// TwinCAT 3 PLC project WinchCylControl
// ProgramVersion: 3.1.4023.0
// libraries:
//   Tc2_Standard, * (Beckhoff Automation GmbH)
//   Tc2_System, * (Beckhoff Automation GmbH)
//   Tc3_Module, * (Beckhoff Automation GmbH)
// project tree:
//   FunctionBlocks/ FB_Encoder.TcPOU, FB_JoystickInputScaling.TcPOU, FB_ValveOutput.TcPOU
//   Inputs/ G_InputList.TcGVL, ST_ControlBoxInputs.TcDUT, ST_CylinderInputs.TcDUT, ST_JoystickScaling.TcDUT, ST_WinchInputs.TcDUT
//   MotionControl/ Path_signal_gen.TcPOU, P_MotionxControl.TcPOU
//   MotionControl/PID-Controllers/ Closed.TcPOU, Open0.TcPOU
//   MotionControl/Structs/ ST_MotionParameters.TcDUT, ST_Params.TcDUT, ST_PathParameters.TcDUT, ST_ValveDeadBand.TcDUT
//   Outputs/ G_OutputList.TcGVL, ST_ValveOutputs.TcDUT
//   / PlcTask.TcTTO
//   POUs/ MAIN.TcPOU
//   Scaling/FBs/ FB_FlowScale.TcPOU, FB_PressureScale.TcPOU
//   Scaling/ G_ScaledIOs.TcGVL, P_Scaling.TcPOU
//   Scaling/Structs/ ST_FlowScale.TcDUT, ST_ScaledCylinderInputs.TcDUT, ST_ScaledWinchInputs.TcDUT
// real-time tasks:
//   TASK PlcTask: cycle T#10ms, priority 20, ADS port 350

CONFIGURATION WinchCylControl
    RESOURCE PLC ON TwinCAT3
        TASK PlcTask(INTERVAL := T#10ms, PRIORITY := 20);
        PROGRAM MAIN WITH PlcTask : MAIN;
    END_RESOURCE
END_CONFIGURATION

// ---- Inputs/ST_ControlBoxInputs.TcDUT
TYPE ST_ControlBoxInputs :
STRUCT
	bAutoMode AT %I* : BOOL;
	bManualMode AT %I*: BOOL;
	bStartButton AT %I*: BOOL;
	bStopButton AT %I* : BOOL; 
	bTopSwitch AT %I*: BOOL; 
	nJoyX : INT;
	nJoyY : INT; 
END_STRUCT
END_TYPE

// ---- Inputs/ST_CylinderInputs.TcDUT
TYPE ST_CylinderInputs :
STRUCT
	fPistonPressure : INT;
	fRodPressure : INT; 
	fCylinderPosition : LREAL; 
END_STRUCT
END_TYPE

// ---- Inputs/ST_JoystickScaling.TcDUT
TYPE ST_JoystickScaling :
STRUCT
	fMaxInputVal : LREAL := 20509.0;
	fMinInputVal : LREAL := 11787.0; 
	fNeutralInputVal : LREAL := 16175.0;
	fNeutralDeadBand : LREAL := 50.0; 
	fMaxOutputVal : LREAL := 1.0;
	fMinOutputVal : LREAL := -1.0;
	fNeutralOutputVal : LREAL := 0.0;
END_STRUCT
END_TYPE

// ---- Inputs/ST_WinchInputs.TcDUT
TYPE ST_WinchInputs :
STRUCT
	fWinchInletPressure : INT;
	fWinchInletPressureSensor : INT;
	fWinchOutletPressure : INT;
	fWinchOutletPressureB1 : INT;
	fWinchDrainPressure : INT; // 40 BAR
	fWinchInletFlow : INT; 
END_STRUCT
END_TYPE

// ---- MotionControl/Structs/ST_MotionParameters.TcDUT
TYPE ST_MotionParameters :
STRUCT
	bClosedLoopStart : BOOL; 
	bOpenLoopStart : BOOL; 
	bWinchEnable : BOOL;
	bCylinderEnable : BOOL; 
END_STRUCT
END_TYPE

// ---- MotionControl/Structs/ST_Params.TcDUT
TYPE ST_Params :
STRUCT
	fEncoderOffset : LREAL := 17574.8; 
	fGBtoDrumScaling : LREAL := 0.000744309; 
END_STRUCT
END_TYPE

// ---- MotionControl/Structs/ST_PathParameters.TcDUT
TYPE ST_PathParameters :
STRUCT
	x0: LREAL := 0;
	v_0: LREAL := 0;
	x_ref: LREAL := 0.3;
	v_ref: LREAL := 0.15;
	t0: LREAL := 0;
	tRamp: LREAL := 2;
	tWait: LREAL := 2;
END_STRUCT
END_TYPE

// ---- MotionControl/Structs/ST_ValveDeadBand.TcDUT
TYPE ST_ValveDeadBand :
STRUCT
	fPosMax : LREAL := 29490.0;
	fPosMin : LREAL := 20950.0;
	fNegMax : LREAL := 18250.0;
	fNegMin : LREAL := 9830.0;
END_STRUCT
END_TYPE

// ---- Outputs/ST_ValveOutputs.TcDUT
TYPE ST_ValveOutputs :
STRUCT
	bEnable AT %I* : BOOL;
	nValveOut AT %Q* : INT;
END_STRUCT
END_TYPE

// ---- Scaling/Structs/ST_FlowScale.TcDUT
TYPE ST_FlowScale :
STRUCT
	fMaxInputValue :LREAL := 32295.0;
 	fMinInputValue :LREAL := 0.0;
 	fNeutralInputValue :LREAL := 15450;
 	fNeutralDeadband :LREAL := 50.0;
	fMaxOutputValue :LREAL := 150.0; 
	fMinOutputValue :LREAL := -150.0; 
	fNeutralOutputValue :LREAL := 0.0; 
END_STRUCT
END_TYPE

// ---- Scaling/Structs/ST_ScaledCylinderInputs.TcDUT
TYPE ST_ScaledCylinderInputs :
STRUCT
	fPistonPressureS : LREAL;
	fRodPressureS : LREAL; 
	fCylinderPositionS : LREAL; 
END_STRUCT
END_TYPE

// ---- Scaling/Structs/ST_ScaledWinchInputs.TcDUT
TYPE ST_ScaledWinchInputs :
STRUCT
	fWinchInletPressureS : LREAL;
	fWinchInletPressureSensorS : LREAL;
	fWinchOutletPressureS : LREAL;
	fWinchOutletPressureB1S : LREAL;
	fWinchDrainPressureS : LREAL; // 40 BAR
	fWinchInletFlowS : LREAL; 
END_STRUCT
END_TYPE

// ---- Inputs/G_InputList.TcGVL
{attribute 'qualified_only'}
VAR_GLOBAL
	
	stModeSelect : ST_ControlBoxInputs; 
	//bManualSelect : BOOL := ST_ControlBoxInputs.bManualMode;
	//bAutoSelect : BOOL := ST_ControlBoxInputs.bAutoMode;
	//bStart : BOOL := ST_ControlBoxInputs.bStartButton;
	//bStop : BOOL := ST_ControlBoxInputs.bStopButton;
	//bTopSwitchToggle : BOOL := ST_ControlBoxInputs.bTopSwitch;

	// Joystick
	stJoystick : ST_ControlBoxInputs; 
	//nJoyXPos : INT := ST_ControlBoxInputs.nJoyX;
	//nJoyYPos : INT := ST_ControlBoxInputs.nJoyY;

	// Cylinder, Winch and pressure inputs
	fSupplyPressure AT %Q* : LREAL;
	fReturnPressure AT %Q*: LREAL;  // 40 BAR
	
	stWinchPressure : ST_WinchInputs;
	//fWinchPressureIn AT %Q* : LREAL := ST_WinchInputs.fWinchInletPressure; // A
	//fWinchPressureSensor AT %Q* : LREAL := ST_WinchInputs.fWinchInletPressureSensor; // A1
 	//fWinchPressureOut AT %Q* : LREAL := ST_WinchInputs.fWinchOutletPressure; // B
	//fWinchPressureOutB1 AT %Q* : LREAL := ST_WinchInputs.fWinchOutletPressureB1; // B1
	
	stCylinderPressures : ST_CylinderInputs;
	//fRodSidePressure AT %Q* : LREAL := ST_CylinderInputs.fRodPressure; 
	//fBoreSidePressure AT %Q* : LREAL := ST_CylinderInputs.fPistonPressure; 
	
	// Flows
	//fWinchFlow AT %Q* : LREAL := ST_WinchInputs.fWinchInletFlow;  
	
	// Får errors her
	
END_VAR

// ---- Outputs/G_OutputList.TcGVL
{attribute 'qualified_only'}
VAR_GLOBAL
	stValveOutWinch : ST_ValveOutputs;
	stValveOutCyl : ST_ValveOutputs; 
END_VAR

// ---- Scaling/G_ScaledIOs.TcGVL
{attribute 'qualified_only'}
VAR_GLOBAL
	scaledJoyX : LREAL; 
	scaledJoyY : LREAL; 
	scaledValve : LREAL; // Valve output based on joystick input [-1...1] 1 = 29490.0, -1 = 9830
	fLoadPosition : LREAL; 
	fWinchInputsScaled : ST_ScaledWinchInputs; 
	fCylinderInputsScaled : ST_ScaledCylinderInputs; 
END_VAR

// ---- POUs/MAIN.TcPOU
PROGRAM MAIN
VAR
END_VAR

END_PROGRAM

// ---- FunctionBlocks/FB_Encoder.TcPOU
FUNCTION_BLOCK FB_Encoder
VAR_INPUT
	nRawInput : UDINT;
	stParam : ST_Params; 
END_VAR
VAR_OUTPUT
	fPosition : LREAL; 
END_VAR
VAR PERSISTENT
	nRounds : DINT;
	nRawLast : DINT;
END_VAR
VAR
	nInput : DINT;
	nTempInputDiff : DINT;
	nCount : DINT;
	nMaxValue30bit : DINT := 1073741823;
	nThreshold30Bit : DINT := nMaxValue30bit/2;
	fScale16bit : LREAL := 360.0/65535.0;
	fTempPos : LREAL; 
END_VAR

nInput := UDINT_TO_DINT(nRawInput);

nTempInputDiff := nInput - nRawLast;

IF (nTempInputDiff > nThreshold30Bit) THEN
	nRounds := nRounds -1;
END_IF

IF (nTempInputDiff < nThreshold30Bit) THEN
	nRounds := nRounds + 1;
END_IF

nCount := nInput + nRounds*nMaxValue30bit;

fPosition := DINT_TO_LREAL(nCount)*fScale16bit - stParam.fEncoderOffset;

END_FUNCTION_BLOCK

// ---- FunctionBlocks/FB_JoystickInputScaling.TcPOU
FUNCTION_BLOCK FB_JoystickInputScaling
VAR_INPUT
	bEnable : BOOL; // Start Button
	bSwitch : BOOL; // TopSwitch
	nRawInput : INT;
	stJoyInputScaling : ST_JoystickScaling; 
	
END_VAR
VAR_OUTPUT
	fNormOutputC : LREAL; // Scaled cylinder output
	fNormOutputW : LREAL; // Scaled winch output
END_VAR
VAR
	fRawInput : LREAL;
	fTempInput : LREAL;
	fTempOutput : LREAL; 
END_VAR

fRawInput := INT_TO_LREAL(nRawInput);

fTempInput := fRawInput - stJoyInputScaling.fNeutralInputVal; 

IF fTempInput > stJoyInputScaling.fNeutralDeadBand THEN
	fTempOutput := fTempInput/(stJoyInputScaling.fMaxInputVal - stJoyInputScaling.fNeutralInputVal);
ELSIF fTempInput < -stJoyInputScaling.fNeutralDeadBand THEN
	fTempOutput := fTempInput/(stJoyInputScaling.fNeutralInputVal - stJoyInputScaling.fMinInputVal); 
ELSE
	fTempOutput := 0.0;
END_IF

IF NOT (bEnable) THEN
	fNormOutputC := 0; // If startbutton is not held, no joystick output
	fNormOutputW := 0.0;
ELSIF bEnable AND NOT bSwitch THEN
	fNormOutputC := LIMIT(stJoyInputScaling.fMinOutputVal, fTempOutput, stJoyInputScaling.fMaxOutputVal); 
	fNormOutputW := 0.0; // If startbutton is held but no top switch, cylinder gets output
ELSE
	fNormOutputC := 0.0; // If startbutton AND topswitch, winch gets output
	fNormOutputW := LIMIT(stJoyInputScaling.fMinOutputVal, fTempOutput, stJoyInputScaling.fMaxOutputVal); 
END_IF

END_FUNCTION_BLOCK

// ---- FunctionBlocks/FB_ValveOutput.TcPOU
FUNCTION_BLOCK FB_ValveOutput
VAR_INPUT
	bEnable : BOOL; 
	bDeadBandCompOn : BOOL;
	stValveDeadBand : ST_ValveDeadBand;
	fNormInput : LREAL; 
END_VAR
VAR_OUTPUT
	bEnableValveOutput : BOOL;
	nOutput : INT;
END_VAR
VAR
	nOffset : INT := 19660;
	nMaxValue : INT := 29490;
	nMinValue : INT := 9830;
	nTempOutput : INT; 
END_VAR

IF bDeadBandCompOn THEN
	IF fNormInput > 0.0 THEN
		nTempOutput := LREAL_TO_INT(ABS(fNormInput*(stValveDeadBand.fPosMax - stValveDeadBand.fPosMin) + stValveDeadBand.fPosMin)); 
	ELSIF fNormInput < 0.0 THEN
		nTempOutput := LREAL_TO_INT(fNormInput*(stValveDeadBand.fNegMax - stValveDeadBand.fNegMin) - stValveDeadBand.fNegMin);
	ELSE
		nTempOutput := nOffset; 
	END_IF
	
ELSE
	IF fNormInput > 0.0 THEN
		nTempOutput := LREAL_TO_INT(ABS(fNormInput*(32767.0 - 19660.0) + 19660.0));
	ELSIF fNormInput < 0.0 THEN
		nTempOutput := LREAL_TO_INT(ABS(fNormInput*(0-19660.0) - 19660.0));
	ELSE
		nTempOutput := nOffset;		
	END_IF
END_IF

IF bEnable THEN
	nOutput := LIMIT(nMinValue, nTempOutput, nMaxValue);
	bEnableValveOutput := TRUE;
ELSE
	nOutput := nOffset;
	bEnableValveOutput := FALSE; 
END_IF

END_FUNCTION_BLOCK

// ---- MotionControl/Path_signal_gen.TcPOU
FUNCTION_BLOCK Path_signal_gen
VAR_INPUT
	x0: LREAL;
	v_0: LREAL;
	x_ref: LREAL;
	v_ref: LREAL;
	t0: LREAL;
	tRamp: LREAL;
	tWait: LREAL;
	t: LREAL;
END_VAR
VAR_OUTPUT
	x: LREAL;
	v: LREAL;
	Error: LREAL;
END_VAR
VAR
	Error_0: DINT;
	tHold: LREAL;
	x1: LREAL;
	x4: LREAL;
	a_tmp: LREAL;
	a_tmp_tmp: LREAL;
	a_tmp_0: LREAL;
	a_tmp_tmp_0: LREAL;
	a_tmp_tmp_1: LREAL;
	a_tmp_tmp_2: LREAL;
	x1_tmp: LREAL;
	x4_tmp: LREAL;
END_VAR


(* MATLAB Function: '<Root>/Path_signal_gen' *)
(* MATLAB Function 'Path_signal_gen': '<S1>:1' *)
(* '<S1>:1:3' x_SetPoint = x_ref - x0; *)
(* '<S1>:1:4' vs = v_ref; *)
(* '<S1>:1:5' slopeExt = v_0-vs; *)
(* '<S1>:1:6' slopeRetr = -vs-v_0; *)
(* '<S1>:1:8' as = vs/tRamp; *)
(* Find acceleration *)
(* '<S1>:1:9' s_acc = (vs^2-v_0^2)/as; *)
(* Acceleration sp *)
(* '<S1>:1:11' tHold = (x_SetPoint-s_acc)/vs; *)
tHold := ((x_ref - x0) - (((v_ref * v_ref) - (v_0 * v_0)) / (v_ref / tRamp))) / v_ref;
(* '<S1>:1:13' if tHold < 0 *)

IF tHold < 0.0 THEN 
    (* '<S1>:1:14' Error = 1; *)
    Error_0 := 1;
ELSE 
    (* '<S1>:1:15' else *)
    (* '<S1>:1:16' Error = 0; *)
    Error_0 := 0;
END_IF;

(* '<S1>:1:19' t1 = tRamp; *)
(* '<S1>:1:20' t2 = tHold; *)
(* '<S1>:1:21' t3 = tRamp; *)
(* '<S1>:1:22' t4 = tWait; *)
(* '<S1>:1:23' t5 = t1; *)
(* '<S1>:1:24' t6 = t2; *)
(* '<S1>:1:25' t7 = t3; *)
(* Ramp Equations: *)
(* '<S1>:1:28' x1 = x0 + v_0*((t0+t1)-t0) - (slopeExt/t1)*((t0+t1)-t0)^2/2; *)
a_tmp_tmp := t0 + tRamp;
a_tmp := a_tmp_tmp - t0;
x1_tmp := (v_0 - v_ref) / tRamp;
x1 := ((a_tmp * v_0) + x0) - ((x1_tmp * (a_tmp * a_tmp)) / 2.0);
(* '<S1>:1:29' x2 = x1 + vs * ((t0+t1+t2)-(t0+t1)); *)
(* '<S1>:1:30' x4 = x_ref - v_0 * ((t0+t1+t2+t3+t4+t5)-(t0+t1+t2+t3+t4)) + (slopeRetr/t5)*((t0+t1+t2+t3+t4+t5)-(t0+t1+t2+t3+t4))^2/2; *)
a_tmp_tmp_0 := a_tmp_tmp + tHold;
a_tmp_tmp_1 := a_tmp_tmp_0 + tRamp;
a_tmp := a_tmp_tmp_1 + tWait;
a_tmp_tmp_2 := a_tmp + tRamp;
a_tmp_0 := a_tmp_tmp_2 - a_tmp;
x4_tmp := (( -v_ref) - v_0) / tRamp;
x4 := (x_ref - (a_tmp_0 * v_0)) + ((x4_tmp * (a_tmp_0 * a_tmp_0)) / 2.0);
(* '<S1>:1:31' x5 = x4 - vs*((t0+t1+t2+t3+t4+t5+t6)-(t0+t1+t2+t3+t4+t5)); *)
(* '<S1>:1:33' if Error == 1 *)

IF Error_0 = 1 THEN 
    (* Outport: '<Root>/x' *)
    (* '<S1>:1:34' x = x0; *)
    x := x0;
    (* Outport: '<Root>/v' *)
    (* '<S1>:1:35' v = v_0; *)
    v := v_0;
ELSIF (t >= 0.0) AND (t < t0) THEN 
    (* Outport: '<Root>/x' *)
    (* '<S1>:1:36' elseif t >= 0 && t<t0 *)
    (* '<S1>:1:37' x = x0; *)
    x := x0;
    (* Outport: '<Root>/v' *)
    (* '<S1>:1:38' v = v_0; *)
    v := v_0;
ELSIF (t >= t0) AND (t < a_tmp_tmp) THEN 
    (* '<S1>:1:39' elseif t >= t0 && t < (t0+t1) *)
    (* '<S1>:1:40' x = x0 + v_0*(t-t0) - (slopeExt/t1)*(t-t0)^2/2; *)
    a_tmp := t - t0;
    (* Outport: '<Root>/x' *)
    x := ((a_tmp * v_0) + x0) - ((x1_tmp * (a_tmp * a_tmp)) / 2.0);
    (* Outport: '<Root>/v' *)
    (* '<S1>:1:41' v = v_0 - (slopeExt/t1)*(t-t0); *)
    v := v_0 - (x1_tmp * a_tmp);
ELSIF (t >= a_tmp_tmp) AND (t < a_tmp_tmp_0) THEN 
    (* Outport: '<Root>/x' *)
    (* '<S1>:1:42' elseif t >=(t0+t1) && t < (t0+t1+t2) *)
    (* '<S1>:1:43' x = x1 + vs*(t-(t0+t1)); *)
    x := ((t - a_tmp_tmp) * v_ref) + x1;
    (* Outport: '<Root>/v' *)
    (* '<S1>:1:44' v = vs; *)
    v := v_ref;
ELSIF (t >= a_tmp_tmp_0) AND (t < a_tmp_tmp_1) THEN 
    (* '<S1>:1:45' elseif t>=(t0+t1+t2) && t<(t0+t1+t2+t3) *)
    (* '<S1>:1:46' x = x2 + vs*(t-(t0+t1+t2)) + (slopeExt/t3)*(t-(t0+t1+t2))^2/2; *)
    a_tmp := t - a_tmp_tmp_0;
    (* Outport: '<Root>/x' *)
    x := ((((a_tmp_tmp_0 - a_tmp_tmp) * v_ref) + x1) + (a_tmp * v_ref)) + ((x1_tmp * (a_tmp * a_tmp)) / 2.0);
    (* Outport: '<Root>/v' *)
    (* '<S1>:1:47' v = vs + (slopeExt/t3)*(t-(t0+t1+t2)); *)
    v := (a_tmp * x1_tmp) + v_ref;
ELSIF (t >= a_tmp_tmp_1) AND (t < a_tmp) THEN 
    (* Outport: '<Root>/x' *)
    (* '<S1>:1:48' elseif t >=(t0+t1+t2+t3) && t<(t0+t1+t2+t3+t4) *)
    (* '<S1>:1:49' x = x_ref; *)
    x := x_ref;
    (* Outport: '<Root>/v' *)
    (* '<S1>:1:50' v = v_0; *)
    v := v_0;
ELSIF (t >= a_tmp) AND (t < a_tmp_tmp_2) THEN 
    (* '<S1>:1:51' elseif t>=(t0+t1+t2+t3+t4) && t < (t0+t1+t2+t3+t4+t5) *)
    (* '<S1>:1:52' x = x_ref - v_0*(t-(t0+t1+t2+t3+t4))+(slopeRetr/t5)*(t-(t0+t1+t2+t3+t4))^2/2; *)
    a_tmp := t - a_tmp;
    (* Outport: '<Root>/x' *)
    x := (x_ref - (a_tmp * v_0)) + ((x4_tmp * (a_tmp * a_tmp)) / 2.0);
    (* Outport: '<Root>/v' *)
    (* '<S1>:1:53' v = v_0 + (slopeRetr/t5)*(t-(t0+t1+t2+t3+t4)); *)
    v := (a_tmp * x4_tmp) + v_0;
ELSE 
    x1_tmp := a_tmp_tmp_2 + tHold;

    IF (t >= a_tmp_tmp_2) AND (t < x1_tmp) THEN 
        (* Outport: '<Root>/x' *)
        (* '<S1>:1:54' elseif t>=(t0+t1+t2+t3+t4+t5) && t < (t0+t1+t2+t3+t4+t5+t6) *)
        (* '<S1>:1:55' x = x4 - vs*(t-(t0+t1+t2+t3+t4+t5)); *)
        x := x4 - ((t - a_tmp_tmp_2) * v_ref);
        (* Outport: '<Root>/v' *)
        (* '<S1>:1:56' v = -vs; *)
        v :=  -v_ref;
    ELSIF (t >= x1_tmp) AND (t < (x1_tmp + tRamp)) THEN 
        (* '<S1>:1:57' elseif t >= (t0+t1+t2+t3+t4+t5+t6) && t < (t0+t1+t2+t3+t4+t5+t6+t7) *)
        (* '<S1>:1:58' x = x5 - vs*(t-(t0+t1+t2+t3+t4+t5+t6)) - (slopeRetr/t3)*(t-(t0+t1+t2+t3+t4+t5+t6))^2/2; *)
        a_tmp := t - x1_tmp;
        (* Outport: '<Root>/x' *)
        x := ((x4 - ((x1_tmp - a_tmp_tmp_2) * v_ref)) - (a_tmp * v_ref)) - ((x4_tmp * (a_tmp * a_tmp)) / 2.0);
        (* Outport: '<Root>/v' *)
        (* '<S1>:1:59' v = -vs-(slopeRetr/t3)*(t-(t0+t1+t2+t3+t4+t5+t6)); *)
        v := ( -v_ref) - (a_tmp * x4_tmp);
    ELSE 
        (* Outport: '<Root>/x' *)
        (* '<S1>:1:60' else *)
        (* '<S1>:1:61' x = x0; *)
        x := x0;
        (* Outport: '<Root>/v' *)
        (* '<S1>:1:62' v = v_0; *)
        v := v_0;
    END_IF;

END_IF;

(* Outport: '<Root>/Error' incorporates:
 *  MATLAB Function: '<Root>/Path_signal_gen' *)
Error := DINT_TO_LREAL(Error_0);

END_FUNCTION_BLOCK

// ---- MotionControl/PID-Controllers/Closed.TcPOU
FUNCTION_BLOCK Closed
VAR_INPUT
	Enable: BOOL;
	KpGain: LREAL;
	PosRef: LREAL;
	Pos_feedback: LREAL;
END_VAR
VAR_OUTPUT
	Ctrl_signal_Pos: LREAL;
	PosErr: LREAL;
END_VAR
VAR
END_VAR


(* Outputs for Atomic SubSystem: '<Root>/Closed-loop PosCtrl (Auto)' *)
(* Sum: '<S1>/Sum' *)
PosErr := PosRef - Pos_feedback;
(* Product: '<S1>/Product' *)
Ctrl_signal_Pos := KpGain * PosErr;
(* Saturate: '<S1>/Predefined Saturation' *)

IF Ctrl_signal_Pos > 1.0 THEN 
    Ctrl_signal_Pos := 1.0;
ELSIF Ctrl_signal_Pos < -1.0 THEN 
    Ctrl_signal_Pos := -1.0;
END_IF;

(* End of Saturate: '<S1>/Predefined Saturation' *)


(* Switch: '<S1>/Switch' *)

IF Enable := FALSE THEN 
    (* Outport: '<Root>/Ctrl_signal_Pos' incorporates:
     *  Constant: '<S1>/Constant' *)
    Ctrl_signal_Pos := 0.0;
END_IF;

(* End of Switch: '<S1>/Switch' *)
(* End of Outputs for SubSystem: '<Root>/Closed-loop PosCtrl (Auto)' *)

END_FUNCTION_BLOCK

// ---- MotionControl/PID-Controllers/Open0.TcPOU
FUNCTION_BLOCK Open0
VAR_INPUT
	vel_refms: LREAL;
	Enable_Signal: BOOL;
	QMax_refLMIN: LREAL;
END_VAR
VAR_OUTPUT
	Ctrl_signalms: LREAL;
END_VAR
VAR
	rtb_Switch: LREAL;
END_VAR


(* Outputs for Atomic SubSystem: '<Root>/Open-loop VelControl (Manual)' *)
(* Switch: '<S1>/Switch' incorporates:
 *  Constant: '<S1>/Annulus_Area'
 *  Constant: '<S1>/Boreside_Area'
 *  Product: '<S1>/Product'
 *  Product: '<S1>/Product1' *)

IF vel_refms > 0.0 THEN 
    rtb_Switch := 0.0033183 * vel_refms;
ELSE 
    rtb_Switch := vel_refms * 0.0023562;
END_IF;

(* End of Switch: '<S1>/Switch' *)


(* Switch: '<S1>/Switch1' incorporates:
 *  Constant: '<S1>/Constant'
 *  Gain: '<S1>/UnitConv'
 *  Product: '<S1>/Divide' *)

IF Enable_Signal THEN 
    Ctrl_signalms := (60000.0 * rtb_Switch) / QMax_refLMIN;
ELSE 
    Ctrl_signalms := 0.0;
END_IF;

(* End of Switch: '<S1>/Switch1' *)


(* Saturate: '<S1>/Saturation' *)

IF Ctrl_signalms > 0.05 THEN 
    (* Outport: '<Root>/Ctrl_signal(m//s)' *)
    Ctrl_signalms := 0.05;
ELSIF Ctrl_signalms < -0.05 THEN 
    (* Outport: '<Root>/Ctrl_signal(m//s)' *)
    Ctrl_signalms := -0.05;
END_IF;

(* End of Saturate: '<S1>/Saturation' *)
(* End of Outputs for SubSystem: '<Root>/Open-loop VelControl (Manual)' *)

END_FUNCTION_BLOCK

// ---- MotionControl/P_MotionxControl.TcPOU
PROGRAM P_MotionxControl
VAR
	// Placeholder for the path
	fMyPath : Path_signal_gen(); 
	fPosCtrl : Closed();
	fVelCtrl : Open0(); 
	
	// Starting conditions for cylinder x winch
	stStartingConditions : ST_MotionParameters; 
	
	// Parameter settings for the path (ramp/x0/v0) etc.
	stPathParams : ST_PathParameters;
	
	// Controller tuning
	fKpP : LREAL := 1; 
	
	// Timer to initialize path
	bTimerStart : BOOL := FALSE; 
	myTimer : TON; 
	
	// References for controllers
	fPosRef : LREAL; 
	fVelRef : LREAL; 
	fError : LREAL; 
	fCylinderFeedback : LREAL := ST_CylinderInputs.fCylinderPosition; 
	fWinchFeedBack : LREAL := FB_Encoder.fPosition; 
	
END_VAR


IF stStartingConditions.bCylinderEnable THEN
	bTimerStart := TRUE;
	myTimer(IN := bTimerStart, PT:=T#20S);
	fMyPath(x0:=stPathParams.x0, v_0:=stPathParams.v_0, x_ref:=stPathParams.x_ref, v_ref:=stPathParams.v_ref, t0:=0, 
	tRamp:=stPathParams.tRamp, tWait:=stPathParams.tWait, t:=myTimer);
	
	fPosRef := fMyPath.x;    
	fVelRef := fMyPath.v;
	fError := fMyPath.Error; 
	
	fPosCtrl(Enable := stStartingConditions.bClosedLoopStart, KpGain := fKpP, 
	PosRef := fPosRef, Pos_feedback := fCylinderFeedback(*Feedback*));  
	
	IF myTimer.Q := TRUE THEN
		bTimerStart := FALSE; 
	END_IF
	
END_IF

IF stStartingConditions.bWinchEnable THEN
	bTimerStart := TRUE;
	myTimer(IN := bTimerStart, PT := T#20S); 
	fMyPath(x0:=stPathParams.x0, v_0:=stPathParams.v_0, x_ref:=stPathParams.x_ref, v_ref:=stPathParams.v_ref, t0:=0, 
	tRamp:=stPathParams.tRamp, tWait:=stPathParams.tWait, t:=myTimer);
	
	fPosRef := fMyPath.x;    
	fVelRef := fMyPath.v;
	fError := fMyPath.Error;
	
	fVelCtrl(vel_refms := fVelRef, Enable_Signal := stStartingConditions.bOpenLoopStart, QMax_refLMIN := 150.0); 
	
	IF myTimer.Q := TRUE THEN
		bTimerStart := FALSE; 
	END_IF
	
END_IF

END_PROGRAM

// ---- Scaling/FBs/FB_FlowScale.TcPOU
FUNCTION_BLOCK FB_FlowScale
VAR_INPUT
	nRawInputFlow : INT; 
	stFlowScaling : ST_FlowScale; 
END_VAR
VAR_OUTPUT
	fScaledOutputFlow : LREAL; 
END_VAR
VAR
	fRealRaw : LREAL; 
	fTempIn : LREAL;  
	fTempOut : LREAL; 
	fMaxFlow : LREAL := 150.0;
END_VAR

fRealRaw := INT_TO_LREAL(nRawInputFlow); 

fTempIn := fRealRaw - stFlowScaling.fNeutralInputValue; 

IF fTempIn > stFlowScaling.fNeutralInputValue THEN
	fTempOut := fTempIn/(stFlowScaling.fMaxInputValue - stFlowScaling.fNeutralInputValue);
ELSIF fTempIn < stFlowScaling.fNeutralInputValue THEN
	fTempOut := fTempIn/(stFlowScaling.fNeutralInputValue - stFlowScaling.fMinInputValue);
ELSE
	fTempOut := 0.0;
END_IF

fScaledOutputFlow := LIMIT(stFlowScaling.fMaxOutputValue, fTempOut*fMaxFlow, stFlowScaling.fMinOutputValue);

END_FUNCTION_BLOCK

// ---- Scaling/FBs/FB_PressureScale.TcPOU
FUNCTION_BLOCK FB_PressureScale
VAR_INPUT
	//nRawPressureVal40 : INT; 
	nRawPressureVal400 : INT; 
END_VAR
VAR_OUTPUT
	//fScaledPressureVal40 : LREAL; 
	fScaledPressureVal400 : LREAL; 
END_VAR
VAR
	//fMaxPressure40 : LREAL := 40.0;
	fMaxPressure400 : LREAL := 400.0;
	fMaxInput : REAL := 32767.0; 
END_VAR

//fScaledPressureVal40 := (INT_TO_LREAL(nRawPressureVal40)/fMaxInput) * fMaxPressure40; 

fScaledPressureVal400 := (INT_TO_LREAL(nRawPressureVal400)/fMaxInput) * fMaxPressure400;

END_FUNCTION_BLOCK

// ---- Scaling/P_Scaling.TcPOU
PROGRAM P_Scaling
VAR
	stJoy : ST_JoystickScaling; // Unscaled Input variables from joystick
	stCylinder : ST_CylinderInputs; // Unscaled pressure x flow values (Cylinder)
	stWinch : ST_WinchInputs; // Unscaled pressure x flow values (Winch)
	fValveScaled : LREAL; 
	
	// FBs
	scalePressure : FB_PressureScale; 
	scaleFlow : FB_FlowScale; 
END_VAR


// Scaling pressures
G_ScaledIOs.fCylinderInputsScaled.fRodPressureS := scalePressure(nRawPressureVal400 := stCylinder.fRodPressure);
G_ScaledIOs.fCylinderInputsScaled.fPistonPressureS := scalePressure(nRawPressureVal400 := stCylinder.fPistonPressure); 
G_ScaledIOs.fWinchInputsScaled.fWinchInletPressureS := scalePressure(nRawPressureVal400 := stWinch.fWinchInletPressure);
G_ScaledIOs.fWinchInputsScaled.fWinchInletPressureSensorS := scalePressure(nRawPressureVal400 := stWinch.fWinchInletPressureSensor);
G_ScaledIOs.fWinchInputsScaled.fWinchOutletPressureS := scalePressure(nRawPressureVal400 := stWinch.fWinchOutletPressure);
G_ScaledIOs.fWinchInputsScaled.fWinchOutletPressureB1S := scalePressure(nRawPressureVal400 := stWinch.fWinchOutletPressureB1);

END_PROGRAM
